// TIA Portal project "Elevator" (V15)

(* hardware
DEVICE "S7-1200 station_1"  S7-1200 Station
   slot 0: "Rack_0"  S7-1200 Rack  Rack  V1.0
   slot 1: "PLC_1"  CPU 1215C DC/DC/Rly  6ES7 215-1HG40-0XB0  V4.2
*)

// ===== PLC "PLC_1"  CPU 1215C DC/DC/Rly =====

VAR_GLOBAL   // PLC tag table "Default tag table"
   ""asansor_cagri_F1"" AT %I4.0 : Bool;
   ""kat_cagri_F1"" AT %I4.5 : Bool;
   ""asansor_cagri_F2"" AT %I4.1 : Bool;
   ""kat_cagri_F2"" AT %I4.6 : Bool;
   ""asansor_cagri_F3"" AT %I4.2 : Bool;
   ""kat_cagri_F3"" AT %I4.7 : Bool;
   ""asansor_cagri_F4"" AT %I4.3 : Bool;
   ""kat_cagri_F4"" AT %I5.0 : Bool;
   ""F1_sensor"" AT %I2.3 : Bool;
   ""F2_sensor"" AT %I2.4 : Bool;
   ""F4_sensor"" AT %I2.6 : Bool;
   ""F3_sensor"" AT %I2.5 : Bool;
   ""F5_sensor"" AT %I2.7 : Bool;
   ""asansor_cagri_F5"" AT %I4.4 : Bool;
   ""kat_cagri_F5"" AT %I5.1 : Bool;
   ""acma_tusu"" AT %I5.5 : Bool;
   ""obstacle"" AT %I2.1 : Bool;
   ""overload"" AT %I2.2 : Bool;
   ""kapama_tusu"" AT %I5.7 : Bool;
   ""Motor_Yukari"" AT %Q7.1 : Bool;
   ""Motor_Asagi"" AT %Q7.2 : Bool;
   ""kapi_motoru"" AT %Q7.0 : Bool;
END_VAR